Staubli VAL3: buildList.pgx

program buildList(num x_nViewMode (dimensions=1))
  local num i
  local string l_sEvent
  local string l_sTemp
  local string l_sId
  local string l_sName
  local bool l_bStatus
  local bool l_bActive
  local string l_sEmpty
  local num l_nSizeOut
  local num l_nSizeIn
  local string l_sMessage
begin
  // INIT the list
  l_sEmpty=""
  l_nSizeOut=-1
  l_nSizeIn=-1
  call out:getSize(l_nSizeOut)
  call in:getSize(l_nSizeIn)
  call use:stringCopy(l_sEmpty,sList)
  // set the view
  switch x_nViewMode
    case 0
      //
      // output
      //
      sMode="OUT"
      for i=0 to l_nSizeOut-1
        // get
        call out:get(l_sId,i)
        call out:isActive(l_bActive,l_sId)
        if l_bActive
          call out:getStatus(l_bStatus,l_sId)
          call use:showBoolStatus(l_bStatus,l_sTemp)
          call out:getItem(l_sName,l_sId)
          call out:isEnable(l_bStatus,l_sId)
          if l_bStatus
            call listAdd(l_sTemp+" "+l_sId+" {"+l_sName+"}")
          else
            call listAdd(l_sTemp+"!"+l_sId+" {"+l_sName+"}")
          endIf
          // SET THE START_STOP_END_HOME
          if l_sName=="start"
            saveData:sOutStart=l_sId
          elseIf l_sName=="stop"
            saveData:sOutStop=l_sId
          elseIf l_sName=="end"
            saveData:sOutEnd=l_sId
          elseIf l_sName=="home"
            saveData:sOutHome=l_sId
          endIf
        endIf
      endFor
    break
    case 1
      //
      // INPUT
      //
      sMode="IN"
      for i=0 to l_nSizeIn-1
        // CS8
        call in:get(l_sId,i)
        call in:isActive(l_bActive,l_sId)
        if l_bActive
          call in:getStatus(l_bStatus,l_sId)
          call use:showBoolStatus(l_bStatus,l_sTemp)
          call in:getItem(l_sName,l_sId)
          call in:isEnable(l_bStatus,l_sId)
          if l_bStatus
            call listAdd(l_sTemp+" "+l_sId+" {"+l_sName+"}")
          else
            call listAdd(l_sTemp+"!"+l_sId+" {"+l_sName+"}")
          endIf
          // SET THE START_STOP_END_HOME
          if l_sName=="start"
            saveData:sInStart=l_sId
          elseIf l_sName=="stop"
            saveData:sInStop=l_sId
          elseIf l_sName=="end"
            saveData:sInEnd=l_sId
          elseIf l_sName=="home"
            saveData:sInHome=l_sId
          endIf
        endIf
      endFor
    break
  endSwitch
  // rebuild the Function LIST
  call use:listempty()
  call use:listadd(sList)
end
